FUNCTION_BLOCK DEV_MGR (* Device Management Service Interface *)
  (* Standard: 61499 Demo ITA *)
  (* Version 0.3, 2007-10-10, JHC, Holobloc Inc, Moved to fb.rt. *)
  (* Version 0.2, 2000-07-24, JHC, Rockwell Automation, Simplified for XML encoding. *)
  (* Version 0.1, 2000-05-16, JHC, Rockwell Automation, File type changed to ".fbt" *)
  (* Version 0.0, 2000-03-19, JHC, Rockwell Automation *)
  (* Compiler header: package fb.rt; *)
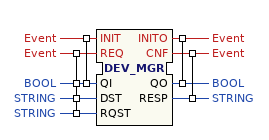
  EVENT_INPUT
    INIT WITH QI; (* Service Initialization/Termination *)
    REQ WITH QI, DST, RQST; (* Service Request *)
  END_EVENT
  EVENT_OUTPUT
    INITO WITH QO; (* Initialization/Termination Confirm *)
    CNF WITH RESP; (* Service Confirmation *)
  END_EVENT
  VAR_INPUT
    QI : BOOL; (* Event Input Qualifier *)
    DST : STRING; (* Destination for RQST *)
    RQST : STRING; (* XML-encoded Request *)
  END_VAR
  VAR_OUTPUT
    QO : BOOL; (* Event Output Qualifier *)
    RESP : STRING; (* XML-encoded Response *)
  END_VAR
  SERVICE DEV_MGR/manager
    SEQUENCE normal_establishment
      DEV_MGR.INIT+() -> manager.init() -> DEV_MGR.INITO+();
    END_SEQUENCE
    SEQUENCE unsuccessful_establishment
      DEV_MGR.INIT+() -> manager.init() -> DEV_MGR.INITO-();
    END_SEQUENCE
    SEQUENCE normal_request
      DEV_MGR.REQ+(RQST) -> manager.serviceRequest(RQST) -> DEV_MGR.CNF+(RESP);
    END_SEQUENCE
    SEQUENCE request_inhibited
      DEV_MGR.REQ-() -> DEV_MGR.CNF-();
    END_SEQUENCE
    SEQUENCE application_initiated_termination
      DEV_MGR.INIT-() -> manager.terminate() -> DEV_MGR.INITO-();
    END_SEQUENCE
    SEQUENCE device_initiated_termination
      manager.terminated() -> DEV_MGR.INITO-();
    END_SEQUENCE
  END_SERVICE
END_FUNCTION_BLOCK
